% RSLogix 500 project 6-2.RSS, saved by version 12.00.00.00 %
PROJECT "UNTITLED"    % processor: Bul.1763 MicroLogix 1100 Series B %

PROGRAM FILES
  LAD 2   10 rungs

DATA FILES
  O0 OUTPUT  5 elements
  I1 INPUT  6 elements
  S2 STATUS  66 elements
  B3 BINARY  1 elements
  T4 TIMER  3 elements
  C5 COUNTER  2 elements
  R6 CONTROL  1 elements
  N7 INTEGER  1 elements
  F8 FLOAT  1 elements

LADDER 2
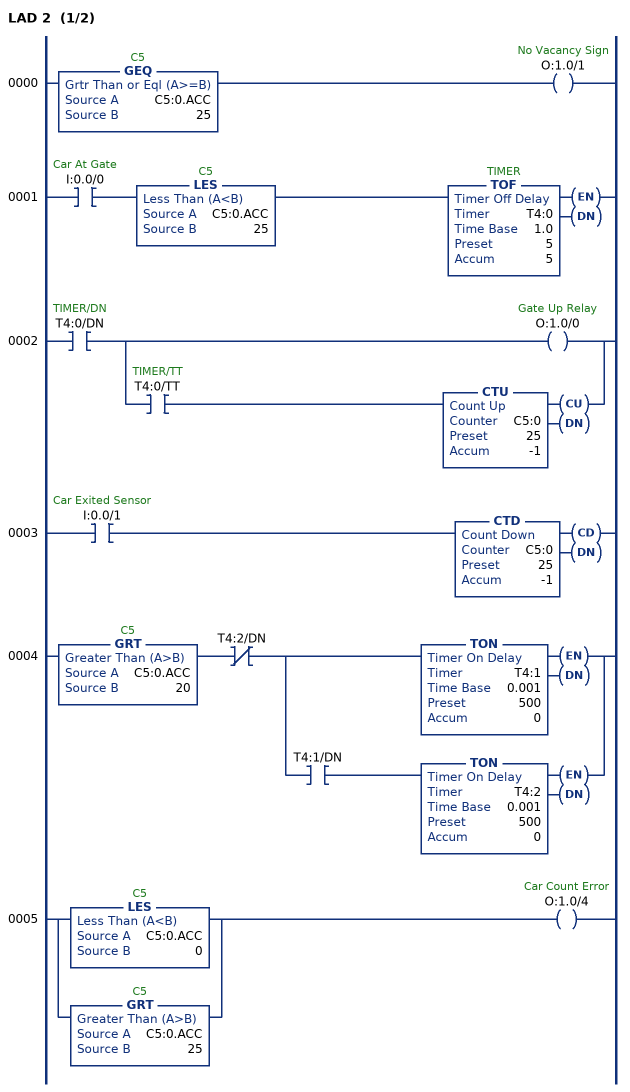
% Rung: 0 %
SOR GEQ C5:0.ACC 25 OTE O:1.0/1 EOR
%   C5:0.ACC  C5 %
%   O:1.0/1  "No Vacancy Sign" %
% Rung: 1 %
SOR XIC I:0.0/0 LES C5:0.ACC 25 TOF T4:0 1.0 5 5 EOR
%   I:0.0/0  "Car At Gate" %
%   C5:0.ACC  C5 %
%   T4:0  TIMER %
% Rung: 2 %
SOR XIC T4:0/DN BST OTE O:1.0/0 NXB XIC T4:0/TT CTU C5:0 25 -1 BND EOR
%   T4:0  TIMER %
%   O:1.0/0  "Gate Up Relay" %
% Rung: 3 %
SOR XIC I:0.0/1 CTD C5:0 25 -1 EOR
%   I:0.0/1  "Car Exited Sensor" %
% Rung: 4 %
SOR GRT C5:0.ACC 20 XIO T4:2/DN BST TON T4:1 0.001 500 0 NXB XIC T4:1/DN TON T4:2 0.001 500 0 BND EOR
%   C5:0.ACC  C5 %
% Rung: 5 %
SOR BST LES C5:0.ACC 0 NXB GRT C5:0.ACC 25 BND OTE O:1.0/4 EOR
%   C5:0.ACC  C5 %
%   O:1.0/4  "Car Count Error" %

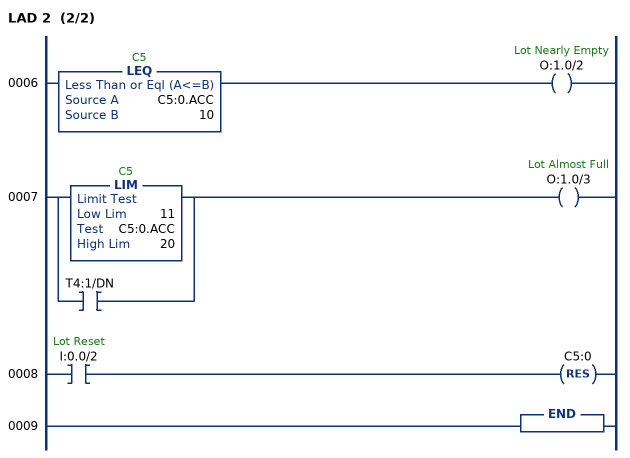
% Rung: 6 %
SOR LEQ C5:0.ACC 10 OTE O:1.0/2 EOR
%   C5:0.ACC  C5 %
%   O:1.0/2  "Lot Nearly Empty" %
% Rung: 7 %
SOR BST LIM 11 C5:0.ACC 20 NXB XIC T4:1/DN BND OTE O:1.0/3 EOR
%   C5:0.ACC  C5 %
%   O:1.0/3  "Lot Almost Full" %
% Rung: 8 %
SOR XIC I:0.0/2 RES C5:0 EOR
%   I:0.0/2  "Lot Reset" %
% Rung: 9 %
SOR END EOR

OTHER DOCUMENTED ADDRESSES
  C5:1  MOV

DATA TABLE (non-zero values as saved)
DATA T4
% .PRE .ACC %
% T4:0 % 5 5
% T4:1 % 500 0
% T4:2 % 500 0
DATA C5
% .PRE .ACC %
% C5:0 % 25 -1
